(* CODESYS project SecadoCafe_ModbusV1.project

Project tree, tasks and I/O mapping:
  Device : CODESYS Control Win V3, 3S - Smart Software Solutions GmbH, order no. 305021, version 3.5.9.10
    application Application
      libraries: Standard, * (System)
      task MainTask (cyclic, interval t#20ms, priority 1) calls PLC_PRG, FLUID_SIIM
      task VISU_TASK (cyclic, interval 100 ms, priority 31) calls VisuElems.Visu_Prg
      task TrendRecordingTask (cyclic, interval 100 ms, priority 31) calls VisuTrendStorageAccess.GlobalInstances.g_TrendRecordingManager.CyclicCall
      program PLC_PRG [ST]
      data type U_WORDS_TO_REAL
      visualisation HMI
      Trend Recording Manager
        HMI_Trend1
      Symbols
      program FLUID_SIIM [LD]
      global variables GVL
    Ethernet : Ethernet, 3S - Smart Software Solutions GmbH, version 3.5.15.0
        settings: IPAddress = [192,168,0,17]; SubnetMask = [255,255,255,0]; GatewayAddress = [192,168,0,1]; MACAddress = [16#7C,16#8A,16#E1,16#B0,16#D0,16#05]; NetworkInterfaceName = 'Ethernet'; NetworkInterfaceName = "Ethernet"; SaveCommunicationSettings = FALSE
      Modbus_TCP_Master : Modbus TCP Master, 3S - Smart Software Solutions GmbH, version 3.5.15.0
          settings: Socket Timeout = 1000; AutoReconnect = TRUE
        Modbus_TCP_Slave : Modbus TCP Slave, 3S - Smart Software Solutions GmbH, version 3.5.15.0
            settings: Unit-ID = 1; IPAddress = [127, 0, 0, 1]; Port = 5020; T_process_hi.Function Code = 3; T_process_hi.Read Offset = 16#0000; T_process_hi.Read Length = 1; T_process_hi.Write Offset = 0; T_process_hi.Write Length = 0; T_process_hi.Cycle Time = 100; heater_cmd.Function Code = 6; heater_cmd.Read Offset = 0; heater_cmd.Read Length = 0; heater_cmd.Write Offset = 16#0002; heater_cmd.Write Length = 1; heater_cmd.Cycle Time = 100; fan_cmd.Function Code = 6; fan_cmd.Read Offset = 0; fan_cmd.Read Length = 0; fan_cmd.Write Offset = 16#0003; fan_cmd.Write Length = 1; fan_cmd.Cycle Time = 100; T_process_lo.Function Code = 3; T_process_lo.Read Offset = 16#0001; T_process_lo.Read Length = 1; T_process_lo.Write Offset = 0; T_process_lo.Write Length = 0; T_process_lo.Cycle Time = 100; plant_mode.Function Code = 6; plant_mode.Read Offset = 0; plant_mode.Read Length = 0; plant_mode.Write Offset = 16#0006; plant_mode.Write Length = 1; plant_mode.Cycle Time = 100; safety_ok.Function Code = 3; safety_ok.Read Offset = 16#0007; safety_ok.Read Length = 1; safety_ok.Write Offset = 0; safety_ok.Write Length = 0; safety_ok.Cycle Time = 100; RH_ambient_hi.Function Code = 3;
              RH_ambient_hi.Read Offset = 16#0004; RH_ambient_hi.Read Length = 1; RH_ambient_hi.Write Offset = 0; RH_ambient_hi.Write Length = 0; RH_ambient_hi.Cycle Time = 100; RH_ambient_lo.Function Code = 3; RH_ambient_lo.Read Offset = 16#0005; RH_ambient_lo.Read Length = 1; RH_ambient_lo.Write Offset = 0; RH_ambient_lo.Write Length = 0; RH_ambient_lo.Cycle Time = 100; tiempo_proceso_hi.Function Code = 3; tiempo_proceso_hi.Read Offset = 16#000A; tiempo_proceso_hi.Read Length = 1; tiempo_proceso_hi.Write Offset = 0; tiempo_proceso_hi.Write Length = 0; tiempo_proceso_hi.Cycle Time = 100; tiempo_proceso_lo.Function Code = 3; tiempo_proceso_lo.Read Offset = 16#000B; tiempo_proceso_lo.Read Length = 1; tiempo_proceso_lo.Write Offset = 0; tiempo_proceso_lo.Write Length = 0; tiempo_proceso_lo.Cycle Time = 100; M_coffee_hi.Function Code = 3; M_coffee_hi.Read Offset = 16#0008; M_coffee_hi.Read Length = 1; M_coffee_hi.Write Offset = 0; M_coffee_hi.Write Length = 0; M_coffee_hi.Cycle Time = 100; M_coffee_lo.Function Code = 3; M_coffee_lo.Read Offset = 16#0009; M_coffee_lo.Read Length = 1; M_coffee_lo.Write Offset = 0; M_coffee_lo.Write Length = 0; M_coffee_lo.Cycle Time = 100; heartbeat.Function Code = 3; heartbeat.Read Offset = 16#000C; heartbeat.Read Length = 1; heartbeat.Write Offset = 0; heartbeat.Write Length = 0;
              heartbeat.Cycle Time = 100
            input  Application.PLC_PRG.T_process_raw[0] : WORD  // T_process_hi
            output Application.PLC_PRG.heater_cmd : WORD  // heater_cmd
            output Application.PLC_PRG.fan_cmd : WORD  // fan_cmd
            input  Application.PLC_PRG.T_process_raw[1] : WORD  // T_process_lo
            output Application.PLC_PRG.plant_mode : WORD  // plant_mode
            input  Application.PLC_PRG.safety_ok : WORD  // safety_ok
            input  Application.PLC_PRG.RH_ambient_raw[0] : WORD  // RH_ambient_hi
            input  Application.PLC_PRG.RH_ambient_raw[1] : WORD  // RH_ambient_lo
            input  Application.PLC_PRG.tiempo_proceso_raw[0] : WORD  // tiempo_proceso_hi
            input  Application.PLC_PRG.tiempo_proceso_raw[1] : WORD  // tiempo_proceso_lo
            input  Application.PLC_PRG.	M_coffee_raw[0] : WORD  // M_coffee_hi
            input  Application.PLC_PRG	.M_coffee_raw[1] : WORD  // M_coffee_lo
            input  Application.PLC_PRG.heartbeat_actual : WORD  // heartbeat
  libraries: VisuSymbols, 3.5.10.0 (System)
  text list GlobalTextList
*)

// Device/Application/U_WORDS_TO_REAL
TYPE U_WORDS_TO_REAL :
UNION
    words : ARRAY[0..1] OF WORD;
    value : REAL;
END_UNION
END_TYPE

// Device/Application/GVL

VAR_GLOBAL
	INPUT0:BYTE;
	OUTPUT0:BYTE;
END_VAR

// Device/Application/PLC_PRG
PROGRAM PLC_PRG
VAR
    // --- Crudo Modbus (words) que se mapean en IO Mapping ---
    T_process_raw   : ARRAY[0..1] OF WORD;
    RH_ambient_raw  : ARRAY[0..1] OF WORD;
    heater_cmd      : WORD;
    fan_cmd         : WORD;
    plant_mode      : WORD;
    safety_ok       : WORD;

    // --- Conversión a REAL ---
    conv_T          : U_WORDS_TO_REAL;
    conv_RH         : U_WORDS_TO_REAL;
    T_process       : REAL;
    RH_ambient      : REAL;

    // --- Auxiliares para el HMI ---
    heater_on       : BOOL;
    fan_on          : BOOL;
    safety_alarm    : BOOL;

    setpoint        : REAL := 50.0;   // °C, solo para esta prueba
	tiempo_proceso_raw : ARRAY[0..1] OF WORD;  // [0]=tiempo_proceso_hi, [1]=tiempo_proceso_lo
    conv_tiempo         : U_WORDS_TO_REAL;      // el mismo UNION que ya tienes
    tiempo_secado_h     : REAL;
	
	M_coffee_raw : ARRAY[0..1] OF WORD;
	conv_mcoffee  : U_WORDS_TO_REAL;
	M_coffee      : REAL;
	
	heartbeat_actual   : WORD;   // viene del IO Mapping
    heartbeat_anterior : WORD;
    tmr_comm           : TON;
    comm_error         : BOOL;

END_VAR

// --- Conversión T_process (palabra BAJA primero, ver nota abajo) ---
conv_T.words[0] := T_process_raw[1];
conv_T.words[1] := T_process_raw[0];
T_process := conv_T.value;

// --- Conversión RH_ambient (mismo truco) ---
conv_RH.words[0] := RH_ambient_raw[1];
conv_RH.words[1] := RH_ambient_raw[0];
RH_ambient := conv_RH.value;

conv_tiempo.words[0] := tiempo_proceso_raw[1];   // palabra BAJA primero
conv_tiempo.words[1] := tiempo_proceso_raw[0];   // palabra ALTA segundo
tiempo_secado_h := conv_tiempo.value;

conv_mcoffee.words[0] := M_coffee_raw[1];
conv_mcoffee.words[1] := M_coffee_raw[0];
M_coffee := conv_mcoffee.value;
// ------Apaltado de si se quema la planta o el trabajador :D
IF heartbeat_actual <> heartbeat_anterior THEN
    tmr_comm(IN := FALSE);
ELSE
    tmr_comm(IN := TRUE, PT := T#4S);
END_IF
heartbeat_anterior := heartbeat_actual;
comm_error := tmr_comm.Q;

IF comm_error THEN
    heater_cmd := 0;
    fan_cmd := 0;
END_IF

// --- Control mínimo tipo bang-bang, solo para esta prueba ---
IF plant_mode = 0 AND NOT comm_error THEN // RUN, sin pérdida de comunicación
    IF T_process < setpoint THEN
        heater_cmd := 1;
    ELSE 
        heater_cmd := 0;
    END_IF;
ELSE // HOLD o comm_error -> valor seguro
    heater_cmd := 0;
END_IF;

fan_cmd := 0; // por ahora sin lógica propia; lo activamos manual desde un Watch si quieres probarlo

// --- Auxiliares para el HMI ---
heater_on    := (heater_cmd = 1);
fan_on       := (fan_cmd = 1);
safety_alarm := (safety_ok = 0);

END_PROGRAM

// Device/Application/FLUID_SIIM
PROGRAM FLUID_SIIM
VAR
END_VAR

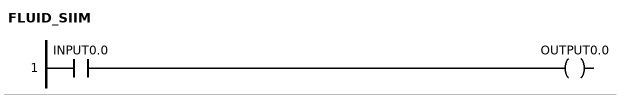
// NETWORK 1
OUTPUT0.0 := INPUT0.0;

END_PROGRAM

// Device/Application/HMI
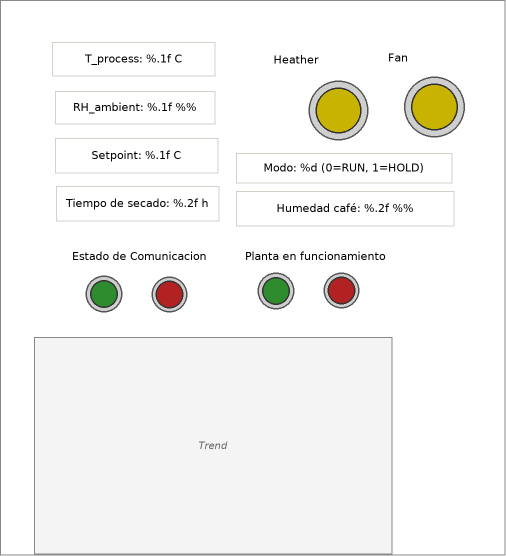
VISUALIZATION HMI  // 506x556
    Textfield (52,42 163x34), "T_process: %.1f C", text variable: PLC_PRG.T_process
    Textfield (55,91 160x33), "RH_ambient: %.1f %%", text variable: PLC_PRG.RH_ambient
    Textfield (55,138 163x35), "Setpoint: %.1f C", text variable: PLC_PRG.setpoint
    Lamp1 (262,76 153x69), variable: PLC_PRG.heater_on, style: Lamp-Lamp1-Yellow
    Lamp1 (365,72 139x70), variable: PLC_PRG.fan_on, style: Lamp-Lamp1-Yellow
    Label (221,47 150x26), "Heather"
    Label (323,45 150x26), "Fan"
    Textfield (236,153 216x30), "Modo: %d (0=RUN, 1=HOLD)", text variable: PLC_PRG.plant_mode
    Lamp1 (319,270 45x41), variable: PLC_PRG.safety_alarm, style: Lamp-Lamp1-Red
    Lamp1 (255,270 42x42), variable: NOT PLC_PRG.safety_alarm, style: Lamp-Lamp1-Green
    Label (184,244 263x25), "Planta en funcionamiento"
    Trend (34,337 358x217)
        p758368661: d
        p2423372160: HH:mm:ss
        p2833066001: HMI_Trend1
    Textfield (56,186 163x35), "Tiempo de secado: %.2f h", text variable: PLC_PRG.tiempo_secado_h
    Textfield (236,191 218x35), "Humedad café: %.2f %%", text variable: PLC_PRG.M_coffee
    Lamp1 (147,274 45x41), variable: PLC_PRG.comm_error, style: Lamp-Lamp1-Red
    Lamp1 (83,273 42x42), variable: NOT PLC_PRG.comm_error, style: Lamp-Lamp1-Green
    Label (8,244 263x25), "Estado de Comunicacion"
END_VISUALIZATION
